FUNCTION_BLOCK EMGYSTOP (* Basic Function Block Type *)
  (* Standard: 61499-2 *)
  (* Version 0.0, 05/07/2022, Etienne, Schneider Electric, Template *)
  PACKAGE Main;
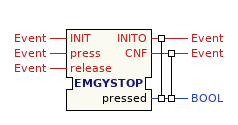
  EVENT_INPUT
    INIT; (* Initialization Request *)
    press; (* Normal Execution Request *)
    release;
  END_EVENT
  EVENT_OUTPUT
    INITO WITH pressed; (* Initialization Confirm *)
    CNF WITH pressed; (* Execution Confirmation *)
  END_EVENT
  VAR_OUTPUT
    pressed : BOOL; (* Output event qualifier *)
  END_VAR
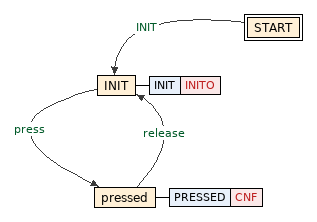
  EC_STATES
    START; (* Initial State *)
    pressed : PRESSED -> CNF;
    INIT : INIT -> INITO;
  END_STATES
  EC_TRANSITIONS
    START TO INIT := INIT;
    INIT TO pressed := press;
    pressed TO INIT := release;
  END_TRANSITIONS
  ALGORITHM INIT IN ST: (* Initialization algorithm *)
;
pressed:=FALSE;
  END_ALGORITHM
  ALGORITHM PRESSED IN ST: (* Normally executed algorithm *)
;
pressed:=TRUE;
  END_ALGORITHM
END_FUNCTION_BLOCK
